{attribute 'qualified_only'}
{attribute 'strict'}
TYPE E_MessageType :
(
	Hint	:= 1,
	Warn	:= 2,
	Error	:= 4
) DWORD;
END_TYPE

// ADSLOG_MSGTYPE_HINT = 1: Message type is hint.
// ADSLOG_MSGTYPE_WARN = 2: Message type is warning.
// ADSLOG_MSGTYPE_ERROR = 4: Message type is error.

(* stored: Version 1.1.0.1, ProductVersion 3.1.4024.11
   EnumerationTextList E_MessageType: Id {a92f99aa-53d2-4b09-8b42-06d9e91f3a85} *)
